PROGRAM MAIN
VAR
END_VAR

END_PROGRAM

(* stored: Version 1.1.0.1
   POU MAIN: Id {99ccac97-1336-465d-a32a-a360f3a1419c} *)
